PROGRAM Stn053_45_CleaningRecircExitDivertRed
VAR
	
	fbTC: FB_CleaningRecircExitDivertTC;
	
//wrong pragma below:
// 		.iMainBufferFull   :=  <0,1,1>TIIB[N47S00 (AL1332)]^N47S03 (AL2341)^TxPDO^input byte 1;

// we are going to use the remote feature instead of linking this
//		.iMainBufferFull   :=  <0,1,0>TIIB[N48S00 (AL1332)]^N48S03 (AL2341)^TxPDO^input byte 2;

	{attribute 'TcLinkToOSO' := '.iPuckPresent   :=  <0,1,0>TIIB[N48S00 (AL1332)]^N48S03 (AL2341)^TxPDO^input byte 0;
		.iDivertMain   :=  <0,1,1>TIIB[N48S00 (AL1332)]^N48S03 (AL2341)^TxPDO^input byte 0;
		.iDivertSpur   :=  <0,1,1>TIIB[N48S00 (AL1332)]^N48S03 (AL2341)^TxPDO^input byte 2;
		.oDivertMain   :=  <0,1,6>TIIB[N48S00 (AL1332)]^N48S02 (EX260)^RxPDO^output byte 2;
		.oDivertSpur   :=  <0,1,7>TIIB[N48S00 (AL1332)]^N48S02 (EX260)^RxPDO^output byte 2;
		.oStopLower   :=  <0,1,3>TIIB[N48S00 (AL1332)]^N48S02 (EX260)^RxPDO^output byte 2'}
	{attribute 'TcLinkTo' := '.fbRFID.iRawArray[0] := TIIB[N48S00 (AL1332)]^N48S04 (DTI425)^TxPDO^input byte 0;
    	.fbRFID.iRawArray[1] := TIIB[N48S00 (AL1332)]^N48S04 (DTI425)^TxPDO^input byte 1;
    	.fbRFID.iRawArray[2] := TIIB[N48S00 (AL1332)]^N48S04 (DTI425)^TxPDO^input byte 2;
    	.fbRFID.iRawArray[3] := TIIB[N48S00 (AL1332)]^N48S04 (DTI425)^TxPDO^input byte 3;
    	.fbRFID.iRawArray[4] := TIIB[N48S00 (AL1332)]^N48S04 (DTI425)^TxPDO^input byte 4;
    	.fbRFID.iRawArray[5] := TIIB[N48S00 (AL1332)]^N48S04 (DTI425)^TxPDO^input byte 5;
    	.fbRFID.iRawArray[6] := TIIB[N48S00 (AL1332)]^N48S04 (DTI425)^TxPDO^input byte 6;
    	.fbRFID.iRawArray[7] := TIIB[N48S00 (AL1332)]^N48S04 (DTI425)^TxPDO^input byte 7;
    	.fbRFID.iRawArray[8] := TIIB[N48S00 (AL1332)]^N48S04 (DTI425)^TxPDO^input byte 8;
    	.fbRFID.iRawArray[9] := TIIB[N48S00 (AL1332)]^N48S04 (DTI425)^TxPDO^input byte 9;
    	.fbRFID.iRawArray[10] := TIIB[N48S00 (AL1332)]^N48S04 (DTI425)^TxPDO^input byte 10;
    	.fbRFID.iRawArray[11] := TIIB[N48S00 (AL1332)]^N48S04 (DTI425)^TxPDO^input byte 11;
    	.fbRFID.iRawArray[12] := TIIB[N48S00 (AL1332)]^N48S04 (DTI425)^TxPDO^input byte 12;
    	.fbRFID.iRawArray[13] := TIIB[N48S00 (AL1332)]^N48S04 (DTI425)^TxPDO^input byte 13;
    	.fbRFID.iRawArray[14] := TIIB[N48S00 (AL1332)]^N48S04 (DTI425)^TxPDO^input byte 14;
    	.fbRFID.iRawArray[15] := TIIB[N48S00 (AL1332)]^N48S04 (DTI425)^TxPDO^input byte 15;
    	.fbRFID.iRawArray[16] := TIIB[N48S00 (AL1332)]^N48S04 (DTI425)^TxPDO^input byte 16;
    	.fbRFID.iRawArray[17] := TIIB[N48S00 (AL1332)]^N48S04 (DTI425)^TxPDO^input byte 17;
    	.fbRFID.iRawArray[18] := TIIB[N48S00 (AL1332)]^N48S04 (DTI425)^TxPDO^input byte 18;
    	.fbRFID.iRawArray[19] := TIIB[N48S00 (AL1332)]^N48S04 (DTI425)^TxPDO^input byte 19;
    	.fbRFID.iRawArray[20] := TIIB[N48S00 (AL1332)]^N48S04 (DTI425)^TxPDO^input byte 20;
    	.fbRFID.iRawArray[21] := TIIB[N48S00 (AL1332)]^N48S04 (DTI425)^TxPDO^input byte 21;
    	.fbRFID.iRawArray[22] := TIIB[N48S00 (AL1332)]^N48S04 (DTI425)^TxPDO^input byte 22;
    	.fbRFID.iRawArray[23] := TIIB[N48S00 (AL1332)]^N48S04 (DTI425)^TxPDO^input byte 23;
    	.fbRFID.iRawArray[24] := TIIB[N48S00 (AL1332)]^N48S04 (DTI425)^TxPDO^input byte 24;
    	.fbRFID.iRawArray[25] := TIIB[N48S00 (AL1332)]^N48S04 (DTI425)^TxPDO^input byte 25;
    	.fbRFID.iRawArray[26] := TIIB[N48S00 (AL1332)]^N48S04 (DTI425)^TxPDO^input byte 26;
    	.fbRFID.iRawArray[27] := TIIB[N48S00 (AL1332)]^N48S04 (DTI425)^TxPDO^input byte 27;
    	.fbRFID.iRawArray[28] := TIIB[N48S00 (AL1332)]^N48S04 (DTI425)^TxPDO^input byte 28;
    	.fbRFID.iRawArray[29] := TIIB[N48S00 (AL1332)]^N48S04 (DTI425)^TxPDO^input byte 29;
    	.fbRFID.iRawArray[30] := TIIB[N48S00 (AL1332)]^N48S04 (DTI425)^TxPDO^input byte 30;
    	.fbRFID.iRawArray[31] := TIIB[N48S00 (AL1332)]^N48S04 (DTI425)^TxPDO^input byte 31;
		.fbRFID.oRawArray[0] := TIIB[N48S00 (AL1332)]^N48S04 (DTI425)^RxPDO^output byte 0;
    	.fbRFID.oRawArray[1] := TIIB[N48S00 (AL1332)]^N48S04 (DTI425)^RxPDO^output byte 1;
    	.fbRFID.oRawArray[2] := TIIB[N48S00 (AL1332)]^N48S04 (DTI425)^RxPDO^output byte 2;
    	.fbRFID.oRawArray[3] := TIIB[N48S00 (AL1332)]^N48S04 (DTI425)^RxPDO^output byte 3;
    	.fbRFID.oRawArray[4] := TIIB[N48S00 (AL1332)]^N48S04 (DTI425)^RxPDO^output byte 4;
    	.fbRFID.oRawArray[5] := TIIB[N48S00 (AL1332)]^N48S04 (DTI425)^RxPDO^output byte 5;
    	.fbRFID.oRawArray[6] := TIIB[N48S00 (AL1332)]^N48S04 (DTI425)^RxPDO^output byte 6;
    	.fbRFID.oRawArray[7] := TIIB[N48S00 (AL1332)]^N48S04 (DTI425)^RxPDO^output byte 7;
    	.fbRFID.oRawArray[8] := TIIB[N48S00 (AL1332)]^N48S04 (DTI425)^RxPDO^output byte 8;
    	.fbRFID.oRawArray[9] := TIIB[N48S00 (AL1332)]^N48S04 (DTI425)^RxPDO^output byte 9;
    	.fbRFID.oRawArray[10] := TIIB[N48S00 (AL1332)]^N48S04 (DTI425)^RxPDO^output byte 10;
    	.fbRFID.oRawArray[11] := TIIB[N48S00 (AL1332)]^N48S04 (DTI425)^RxPDO^output byte 11;
    	.fbRFID.oRawArray[12] := TIIB[N48S00 (AL1332)]^N48S04 (DTI425)^RxPDO^output byte 12;
    	.fbRFID.oRawArray[13] := TIIB[N48S00 (AL1332)]^N48S04 (DTI425)^RxPDO^output byte 13;
    	.fbRFID.oRawArray[14] := TIIB[N48S00 (AL1332)]^N48S04 (DTI425)^RxPDO^output byte 14;
    	.fbRFID.oRawArray[15] := TIIB[N48S00 (AL1332)]^N48S04 (DTI425)^RxPDO^output byte 15;
    	.fbRFID.oRawArray[16] := TIIB[N48S00 (AL1332)]^N48S04 (DTI425)^RxPDO^output byte 16;
    	.fbRFID.oRawArray[17] := TIIB[N48S00 (AL1332)]^N48S04 (DTI425)^RxPDO^output byte 17;
    	.fbRFID.oRawArray[18] := TIIB[N48S00 (AL1332)]^N48S04 (DTI425)^RxPDO^output byte 18;
    	.fbRFID.oRawArray[19] := TIIB[N48S00 (AL1332)]^N48S04 (DTI425)^RxPDO^output byte 19;
    	.fbRFID.oRawArray[20] := TIIB[N48S00 (AL1332)]^N48S04 (DTI425)^RxPDO^output byte 20;
    	.fbRFID.oRawArray[21] := TIIB[N48S00 (AL1332)]^N48S04 (DTI425)^RxPDO^output byte 21;
    	.fbRFID.oRawArray[22] := TIIB[N48S00 (AL1332)]^N48S04 (DTI425)^RxPDO^output byte 22;
    	.fbRFID.oRawArray[23] := TIIB[N48S00 (AL1332)]^N48S04 (DTI425)^RxPDO^output byte 23;
    	.fbRFID.oRawArray[24] := TIIB[N48S00 (AL1332)]^N48S04 (DTI425)^RxPDO^output byte 24;
    	.fbRFID.oRawArray[25] := TIIB[N48S00 (AL1332)]^N48S04 (DTI425)^RxPDO^output byte 25;
    	.fbRFID.oRawArray[26] := TIIB[N48S00 (AL1332)]^N48S04 (DTI425)^RxPDO^output byte 26;
    	.fbRFID.oRawArray[27] := TIIB[N48S00 (AL1332)]^N48S04 (DTI425)^RxPDO^output byte 27;
    	.fbRFID.oRawArray[28] := TIIB[N48S00 (AL1332)]^N48S04 (DTI425)^RxPDO^output byte 28;
    	.fbRFID.oRawArray[29] := TIIB[N48S00 (AL1332)]^N48S04 (DTI425)^RxPDO^output byte 29;
    	.fbRFID.oRawArray[30] := TIIB[N48S00 (AL1332)]^N48S04 (DTI425)^RxPDO^output byte 30;
    	.fbRFID.oRawArray[31] := TIIB[N48S00 (AL1332)]^N48S04 (DTI425)^RxPDO^output byte 31'}
	fbConvDivert: FB_ConvDivertPuck;

	{attribute 'TcLinkToOSO' := '<0,1,2>TIIB[N48S00 (AL1332)]^N48S03 (AL2341)^TxPDO^input byte 2'}
	iSpurBufferFull AT %I*: BOOL;		

END_VAR

//VB13 near Stn 221
//CleaningRecircExit DivertMainPrestopRED  (10B)
//CleaningRecircExit DivertMain (12AB)
//CleaningRecircExitDivertSpur (12AB)
//RED Cleaning Recirc Exit Divert Stop Puck Present (N47S03)
//RED Cleaning Recirc Exit Merge Main Stop DS Buffer  (N48S03)
//RED Cleaning Recirc Exit Diverter Spur
//RED Cleaning Recirc Exit Diverter Main

//RED Cleaning Recirc Exit Divert Spur DS Buffer

// Mappings to/from remote stations
gStn053_45_CleaningRecircExitDivertRed.MainHeartbeatOK := TRUE; // because this PLC is Main
gStn053_45_CleaningRecircExitDivertRed.MainConvRunning :=  gConsumed_SafetyInterfaceConv.MtrRunning.Enc056Mtr07;
gStn053_45_CleaningRecircExitDivertRed.MainInAuto := gStn053.CycleAuto;

gStn053_45_CleaningRecircExitDivertRed.SpurHeartbeatOK := TRUE;
gStn053_45_CleaningRecircExitDivertRed.SpurConvRunning := gConsumed_SafetyInterfaceConv.MtrRunning.Enc056Mtr09;
gStn053_45_CleaningRecircExitDivertRed.SpurInAuto := gStn053.CycleAuto;

gStn053_45_CleaningRecircExitDivertRed.SpurBufferFull := iSpurBufferFull;
gStn053_45_CleaningRecircExitDivertRed.RemoteBufferFullMain := gStn053_47_CleaningRecircExitSpurMergePrestopRed.StatusPuckPresent;

//TODO RCC - Eventually populate station bypass inputs to TC
// Call to traffic control function block.
fbTC(
	pCmp := ADR(gStn053_45_CleaningRecircExitDivertRed)
);
// force stop lower for now. the above is not being populated correctly
// Call to divert component logic instance.
fbConvDivert(
	pStn := ADR(gStn053),
	pCmp := ADR(gStn053_45_CleaningRecircExitDivertRed),
	pStateTraceBuffer := ADR(gStn053_StateTraceBuffer),
	pStateTraceFifo := ADR(gStn053_StateTraceFifo),
	pStats := ADR(gStn053_02_Stats));

END_PROGRAM

(* stored: Version 1.1.0.1, ProductVersion 3.1.4024.6
   POU Stn053_45_CleaningRecircExitDivertRed: Id {e541ad62-5e9c-49b1-9cda-fce8f6c83789}, SpecialFunc None *)
